	// //position fermeture
	// "DB_BIBLIOTHEQUE".Mobile[#index].Pos[0].Entr0_Ap_Pos[0] := "I_RPO_VER_MLG2";
	// "DB_BIBLIOTHEQUE".Mobile[#index].Pos[0].Entr1_Ap_Pos[0] := "I_RPF_VER_MLG2";
	// "DB_BIBLIOTHEQUE".Mobile[#index].Pos[0].Sort0[0] := "I_CO_ver_MLG2";
	// "DB_BIBLIOTHEQUE".Mobile[#index].Pos[0].Sort0_Pr_Fin_Pos[0] := "I_CO_ver_MLG2";

	// //position ouverture
	// "DB_BIBLIOTHEQUE".Mobile[#index].Pos[1].Entr0_Ap_Pos[0] := "I_RPF_VER_MLG2";
	// "DB_BIBLIOTHEQUE".Mobile[#index].Pos[1].Entr1_Ap_Pos[0] := "I_RPO_VER_MLG2";
	// "DB_BIBLIOTHEQUE".Mobile[#index].Pos[1].Sort1[0] := "I_CO_ver_MLG2";
	// "DB_BIBLIOTHEQUE".Mobile[#index].Pos[1].Sort0_Pr_Fin_Pos[0] := "I_CO_ver_MLG2";
	#index := #index + 1;
	//++++++++++++++++++++++++++++++++++++++++++++++++++++++++++++++/*347*/
	"DB_BIBLIOTHEQUE".Mobile[#index].Nom := 'TMEL2';
	"DB_BIBLIOTHEQUE".Mobile[#index].Tjr_Desasservi := TRUE;
	"Init_Tps"(#index);
	#index := #index + 1;
	//++++++++++++++++++++++++++++++++++++++++++++++++++++++++++++++/*348*/
	"DB_BIBLIOTHEQUE".Mobile[#index].Nom := 'BDBP4';
	"DB_BIBLIOTHEQUE".Mobile[#index].Noeud := TRUE;
	"DB_BIBLIOTHEQUE".Mobile[#index].Mob_Suiv[0] := "Index_Mobile"('MLG1');
	"DB_BIBLIOTHEQUE".Mobile[#index].Mob_Suiv[1] := "Index_Mobile"('MLG2');
	"DB_BIBLIOTHEQUE".Mobile[#index].Pos[0].Nom := 'GAUCHE';
	"DB_BIBLIOTHEQUE".Mobile[#index].Pos[0].Mob_Suiv[0] := "Index_Mobile"('MLG2');
	"DB_BIBLIOTHEQUE".Mobile[#index].Pos[1].Nom := 'DROITE';
	"DB_BIBLIOTHEQUE".Mobile[#index].Pos[1].Mob_Suiv[0] := "Index_Mobile"('MLG');
	"DB_BIBLIOTHEQUE".Mobile[#index].Tjr_Desasservi := TRUE;
	"DB_BIBLIOTHEQUE".Mobile[#index].Tps_Att := t#500ms;
	"DB_BIBLIOTHEQUE".Mobile[#index].Tps_Arr := t#0ms;

	//Entrées
	"DB_BIBLIOTHEQUE".Mobile[#index].Pos[0].Entr0_Ap_Pos[0] := "I_RP_BDBP4_MLG2";
	"DB_BIBLIOTHEQUE".Mobile[#index].Pos[0].Entr1_Ap_Pos[0] := "I_RP_BDBP4_MLG1";
	"DB_BIBLIOTHEQUE".Mobile[#index].Pos[0].Sort1[0] := "I_CP_BDBP4_MLG1";
	"DB_BIBLIOTHEQUE".Mobile[#index].Pos[0].Sort0[0] := "I_CP_BDBP4_MLG2";
	"DB_BIBLIOTHEQUE".Mobile[#index].Pos[0].Sort0_Pr_Fin_Pos[0] := "I_CP_BDBP4_MLG1";
	"DB_BIBLIOTHEQUE".Mobile[#index].Pos[0].Sort0_Pr_Fin_Pos[1] := "I_CP_BDBP4_MLG2";


	"DB_BIBLIOTHEQUE".Mobile[#index].Pos[1].Entr0_Ap_Pos[1] := "I_RP_BDBP4_MLG1";
	"DB_BIBLIOTHEQUE".Mobile[#index].Pos[1].Entr1_Ap_Pos[1] := "I_RP_BDBP4_MLG2";

	//Sorties
	"DB_BIBLIOTHEQUE".Mobile[#index].Pos[1].Sort1[0] := "I_CP_BDBP4_MLG2";
	"DB_BIBLIOTHEQUE".Mobile[#index].Pos[1].Sort0[0] := "I_CP_BDBP4_MLG1";
	"DB_BIBLIOTHEQUE".Mobile[#index].Pos[1].Sort0_Pr_Fin_Pos[0] := "I_CP_BDBP4_MLG1";
	"DB_BIBLIOTHEQUE".Mobile[#index].Pos[1].Sort0_Pr_Fin_Pos[1] := "I_CP_BDBP4_MLG2";
	#index := #index + 1;
	//++++++++++++++++++++++++++++++++++++++++++++++++++++++++++++++/*349*/
	"DB_BIBLIOTHEQUE".Mobile[#index].Nom := 'TRP1_TMEL2';
	// "DB_BIBLIOTHEQUE".Mobile[#index].Mob_Suiv[0] := "Index_Mobile"('TMEL');
	"DB_BIBLIOTHEQUE".Mobile[#index].Pos[0].Nom := 'OUVERTURE';
	"DB_BIBLIOTHEQUE".Mobile[#index].Pos[1].Nom := 'FERMETURE';
	"DB_BIBLIOTHEQUE".Mobile[#index].Tjr_Desasservi := TRUE;
	"Init_Tps"(#index);

	//position fermeture
	"DB_BIBLIOTHEQUE".Mobile[#index].Pos[0].Entr0_Ap_Pos[0] := "I_RPO_TRP1_TMEL2";
	"DB_BIBLIOTHEQUE".Mobile[#index].Pos[0].Entr1_Ap_Pos[0] := "I_RPF_TRP1_TMEL2";
	"DB_BIBLIOTHEQUE".Mobile[#index].Pos[0].Sort0[0] := "I_CO_TRP1_TMEL2";
	"DB_BIBLIOTHEQUE".Mobile[#index].Pos[0].Sort0_Pr_Fin_Pos[0] := "I_CO_TRP1_TMEL2";

	//position ouverture
	"DB_BIBLIOTHEQUE".Mobile[#index].Pos[1].Entr0_Ap_Pos[0] := "I_RPF_TRP1_TMEL2";
	"DB_BIBLIOTHEQUE".Mobile[#index].Pos[1].Entr1_Ap_Pos[0] := "I_RPO_TRP1_TMEL2";
	"DB_BIBLIOTHEQUE".Mobile[#index].Pos[1].Sort1[0] := "I_CO_TRP1_TMEL2";
	"DB_BIBLIOTHEQUE".Mobile[#index].Pos[1].Sort0_Pr_Fin_Pos[0] := "I_CO_TRP1_TMEL2";
	#index := #index + 1;

	//++++++++++++++++++++++++++++++//DD01//++++++++++++++++++++++++++++++++/*350*/
	"DB_BIBLIOTHEQUE".Mobile[#index].Noeud := TRUE;


	"DB_BIBLIOTHEQUE".Mobile[#index].Nom := 'DD01';                                  //NOEUD
	"DB_BIBLIOTHEQUE".Mobile[#index].Mob_Suiv[0] := "Index_Mobile"('BV01');
	"DB_BIBLIOTHEQUE".Mobile[#index].Mob_Suiv[1] := "Index_Mobile"('BV02');
	"DB_BIBLIOTHEQUE".Mobile[#index].Mob_Suiv[2] := "Index_Mobile"('BV03');
	"DB_BIBLIOTHEQUE".Mobile[#index].Mob_Suiv[3] := "Index_Mobile"('BV04');
	"DB_BIBLIOTHEQUE".Mobile[#index].Mob_Suiv[4] := "Index_Mobile"('BV05');
	"DB_BIBLIOTHEQUE".Mobile[#index].Mob_Suiv[5] := "Index_Mobile"('BV06');
	"DB_BIBLIOTHEQUE".Mobile[#index].Mob_Prec[0] := "Index_Mobile"('BDE24');


	"DB_BIBLIOTHEQUE".Mobile[#index].Pos[0].Nom := '_BV01';
	"DB_BIBLIOTHEQUE".Mobile[#index].Pos[0].Mob_Suiv[0] := "Index_Mobile"('BV01');
	"DB_BIBLIOTHEQUE".Mobile[#index].Pos[1].Nom := '_BV02';
	"DB_BIBLIOTHEQUE".Mobile[#index].Pos[1].Mob_Suiv[0] := "Index_Mobile"('BV02');
	"DB_BIBLIOTHEQUE".Mobile[#index].Pos[2].Nom := '_BV03';
	"DB_BIBLIOTHEQUE".Mobile[#index].Pos[2].Mob_Suiv[0] := "Index_Mobile"('BV03');
	"DB_BIBLIOTHEQUE".Mobile[#index].Pos[3].Nom := '_BV04';
	"DB_BIBLIOTHEQUE".Mobile[#index].Pos[3].Mob_Suiv[0] := "Index_Mobile"('BV04');
	"DB_BIBLIOTHEQUE".Mobile[#index].Pos[4].Nom := '_BV05';
	"DB_BIBLIOTHEQUE".Mobile[#index].Pos[4].Mob_Suiv[0] := "Index_Mobile"('BV05');
	"DB_BIBLIOTHEQUE".Mobile[#index].Pos[5].Nom := '_BV06';
	"DB_BIBLIOTHEQUE".Mobile[#index].Pos[5].Mob_Suiv[0] := "Index_Mobile"('BV06');

	"Init_Tps"(#index);

	// VERS BV1
	"DB_BIBLIOTHEQUE".Mobile[#index].Pos[0].Entr0_Ap_Pos[0] := "I_RP_DD01_BV2";
	"DB_BIBLIOTHEQUE".Mobile[#index].Pos[0].Entr0_Ap_Pos[1] := "I_RP_DD01_BV3";
	"DB_BIBLIOTHEQUE".Mobile[#index].Pos[0].Entr0_Ap_Pos[2] := "I_RP_DD01_BV4";
	"DB_BIBLIOTHEQUE".Mobile[#index].Pos[0].Entr0_Ap_Pos[3] := "I_RP_DD01_BV5";
	"DB_BIBLIOTHEQUE".Mobile[#index].Pos[0].Entr0_Ap_Pos[4] := "I_RP_DD01_BV6";
	"DB_BIBLIOTHEQUE".Mobile[#index].Pos[0].Entr1_Ap_Pos[0] := "I_RP_DD01_BV1";
	"DB_BIBLIOTHEQUE".Mobile[#index].Pos[0].Sort1[0] := "I_CM_DD01";
	"DB_BIBLIOTHEQUE".Mobile[#index].Pos[0].Sort1[1] := "I_FCP_DD01_BV1";
	"DB_BIBLIOTHEQUE".Mobile[#index].Pos[0].Sort0_Pr_Fin_Pos[0] := "I_CM_DD01";
	"DB_BIBLIOTHEQUE".Mobile[#index].Pos[0].Sort0_Pr_Fin_Pos[1] := "I_FCP_DD01_BV1";
	"DB_BIBLIOTHEQUE".Mobile[#index].Pos[0].Sort0_Ap_Pos[0] := "I_CM_DD01";
	// VERS BV2
	"DB_BIBLIOTHEQUE".Mobile[#index].Pos[1].Entr0_Ap_Pos[0] := "I_RP_DD01_BV1";
	"DB_BIBLIOTHEQUE".Mobile[#index].Pos[1].Entr0_Ap_Pos[1] := "I_RP_DD01_BV3";
	"DB_BIBLIOTHEQUE".Mobile[#index].Pos[1].Entr0_Ap_Pos[2] := "I_RP_DD01_BV4";
	"DB_BIBLIOTHEQUE".Mobile[#index].Pos[1].Entr0_Ap_Pos[3] := "I_RP_DD01_BV5";
	"DB_BIBLIOTHEQUE".Mobile[#index].Pos[1].Entr0_Ap_Pos[4] := "I_RP_DD01_BV6";
	"DB_BIBLIOTHEQUE".Mobile[#index].Pos[1].Entr1_Ap_Pos[0] := "I_RP_DD01_BV2";
	"DB_BIBLIOTHEQUE".Mobile[#index].Pos[1].Sort1[0] := "I_CM_DD01";
	"DB_BIBLIOTHEQUE".Mobile[#index].Pos[1].Sort1[1] := "I_FCP_DD01_BV2";
	"DB_BIBLIOTHEQUE".Mobile[#index].Pos[1].Sort0_Pr_Fin_Pos[0] := "I_CM_DD01";
	"DB_BIBLIOTHEQUE".Mobile[#index].Pos[1].Sort0_Pr_Fin_Pos[1] := "I_FCP_DD01_BV2";
	"DB_BIBLIOTHEQUE".Mobile[#index].Pos[1].Sort0_Ap_Pos[0] := "I_CM_DD01";
	//VERS BV3
	"DB_BIBLIOTHEQUE".Mobile[#index].Pos[2].Entr0_Ap_Pos[0] := "I_RP_DD01_BV1";
	"DB_BIBLIOTHEQUE".Mobile[#index].Pos[2].Entr0_Ap_Pos[1] := "I_RP_DD01_BV2";
	"DB_BIBLIOTHEQUE".Mobile[#index].Pos[2].Entr0_Ap_Pos[2] := "I_RP_DD01_BV4";
	"DB_BIBLIOTHEQUE".Mobile[#index].Pos[2].Entr0_Ap_Pos[3] := "I_RP_DD01_BV5";
	"DB_BIBLIOTHEQUE".Mobile[#index].Pos[2].Entr0_Ap_Pos[4] := "I_RP_DD01_BV6";
	"DB_BIBLIOTHEQUE".Mobile[#index].Pos[2].Entr1_Ap_Pos[0] := "I_RP_DD01_BV3";
	"DB_BIBLIOTHEQUE".Mobile[#index].Pos[2].Sort1[0] := "I_CM_DD01";
	"DB_BIBLIOTHEQUE".Mobile[#index].Pos[2].Sort1[1] := "I_FCP_DD01_BV3";
	"DB_BIBLIOTHEQUE".Mobile[#index].Pos[2].Sort0_Pr_Fin_Pos[0] := "I_CM_DD01";
	"DB_BIBLIOTHEQUE".Mobile[#index].Pos[2].Sort0_Pr_Fin_Pos[1] := "I_FCP_DD01_BV3";
	"DB_BIBLIOTHEQUE".Mobile[#index].Pos[2].Sort0_Ap_Pos[0] := "I_CM_DD01";
	//VERS BV4
	"DB_BIBLIOTHEQUE".Mobile[#index].Pos[3].Entr0_Ap_Pos[0] := "I_RP_DD01_BV1";
	"DB_BIBLIOTHEQUE".Mobile[#index].Pos[3].Entr0_Ap_Pos[1] := "I_RP_DD01_BV2";
	"DB_BIBLIOTHEQUE".Mobile[#index].Pos[3].Entr0_Ap_Pos[2] := "I_RP_DD01_BV3";
	"DB_BIBLIOTHEQUE".Mobile[#index].Pos[3].Entr0_Ap_Pos[3] := "I_RP_DD01_BV5";
	"DB_BIBLIOTHEQUE".Mobile[#index].Pos[3].Entr0_Ap_Pos[4] := "I_RP_DD01_BV6";
	"DB_BIBLIOTHEQUE".Mobile[#index].Pos[3].Entr1_Ap_Pos[0] := "I_RP_DD01_BV4";
	"DB_BIBLIOTHEQUE".Mobile[#index].Pos[3].Sort1[0] := "I_CM_DD01";
	"DB_BIBLIOTHEQUE".Mobile[#index].Pos[3].Sort1[1] := "I_FCP_DD01_BV4";
	"DB_BIBLIOTHEQUE".Mobile[#index].Pos[3].Sort0_Pr_Fin_Pos[0] := "I_CM_DD01";
	"DB_BIBLIOTHEQUE".Mobile[#index].Pos[3].Sort0_Pr_Fin_Pos[1] := "I_FCP_DD01_BV4";
	"DB_BIBLIOTHEQUE".Mobile[#index].Pos[3].Sort0_Ap_Pos[0] := "I_CM_DD01";
	//VERS BV5
	"DB_BIBLIOTHEQUE".Mobile[#index].Pos[4].Entr0_Ap_Pos[0] := "I_RP_DD01_BV1";
	"DB_BIBLIOTHEQUE".Mobile[#index].Pos[4].Entr0_Ap_Pos[1] := "I_RP_DD01_BV2";
	"DB_BIBLIOTHEQUE".Mobile[#index].Pos[4].Entr0_Ap_Pos[2] := "I_RP_DD01_BV3";
	"DB_BIBLIOTHEQUE".Mobile[#index].Pos[4].Entr0_Ap_Pos[3] := "I_RP_DD01_BV4";
	"DB_BIBLIOTHEQUE".Mobile[#index].Pos[4].Entr0_Ap_Pos[4] := "I_RP_DD01_BV6";
	"DB_BIBLIOTHEQUE".Mobile[#index].Pos[4].Entr1_Ap_Pos[0] := "I_RP_DD01_BV5";
	"DB_BIBLIOTHEQUE".Mobile[#index].Pos[4].Sort1[0] := "I_CM_DD01";
	"DB_BIBLIOTHEQUE".Mobile[#index].Pos[4].Sort1[1] := "I_FCP_DD01_BV5";
	"DB_BIBLIOTHEQUE".Mobile[#index].Pos[4].Sort0_Pr_Fin_Pos[0] := "I_CM_DD01";
	"DB_BIBLIOTHEQUE".Mobile[#index].Pos[4].Sort0_Pr_Fin_Pos[1] := "I_FCP_DD01_BV5";
	"DB_BIBLIOTHEQUE".Mobile[#index].Pos[4].Sort0_Ap_Pos[0] := "I_CM_DD01";
	//VERS BV6
	"DB_BIBLIOTHEQUE".Mobile[#index].Pos[5].Entr0_Ap_Pos[0] := "I_RP_DD01_BV1";
	"DB_BIBLIOTHEQUE".Mobile[#index].Pos[5].Entr0_Ap_Pos[1] := "I_RP_DD01_BV2";
	"DB_BIBLIOTHEQUE".Mobile[#index].Pos[5].Entr0_Ap_Pos[2] := "I_RP_DD01_BV3";
	"DB_BIBLIOTHEQUE".Mobile[#index].Pos[5].Entr0_Ap_Pos[3] := "I_RP_DD01_BV4";
	"DB_BIBLIOTHEQUE".Mobile[#index].Pos[5].Entr0_Ap_Pos[4] := "I_RP_DD01_BV5";
	"DB_BIBLIOTHEQUE".Mobile[#index].Pos[5].Entr1_Ap_Pos[0] := "I_RP_DD01_BV6";
	"DB_BIBLIOTHEQUE".Mobile[#index].Pos[5].Sort1[0] := "I_CM_DD01";
	"DB_BIBLIOTHEQUE".Mobile[#index].Pos[5].Sort1[1] := "I_FCP_DD01_BV6";
	"DB_BIBLIOTHEQUE".Mobile[#index].Pos[5].Sort0_Pr_Fin_Pos[0] := "I_CM_DD01";
	"DB_BIBLIOTHEQUE".Mobile[#index].Pos[5].Sort0_Pr_Fin_Pos[1] := "I_FCP_DD01_BV6";
	"DB_BIBLIOTHEQUE".Mobile[#index].Pos[5].Sort0_Ap_Pos[0] := "I_CM_DD01";
	#index := #index + 1;
	//++++++++++++++++++++++++++++++//DD02//++++++++++++++++++++++++++++++++/*351*/
	"DB_BIBLIOTHEQUE".Mobile[#index].Nom := 'DD02';
	"DB_BIBLIOTHEQUE".Mobile[#index].Noeud := TRUE;  //NOEUD
	"DB_BIBLIOTHEQUE".Mobile[#index].Mob_Suiv[0] := "Index_Mobile"('BV07');
	"DB_BIBLIOTHEQUE".Mobile[#index].Mob_Suiv[1] := "Index_Mobile"('BV08');
	"DB_BIBLIOTHEQUE".Mobile[#index].Mob_Suiv[2] := "Index_Mobile"('BV09');
	"DB_BIBLIOTHEQUE".Mobile[#index].Mob_Suiv[3] := "Index_Mobile"('BV10');
	"DB_BIBLIOTHEQUE".Mobile[#index].Mob_Suiv[4] := "Index_Mobile"('BV11');
	"DB_BIBLIOTHEQUE".Mobile[#index].Mob_Suiv[5] := "Index_Mobile"('BV12');
	"DB_BIBLIOTHEQUE".Mobile[#index].Mob_Prec[0] := "Index_Mobile"('T54');

	"DB_BIBLIOTHEQUE".Mobile[#index].Pos[0].Nom := '_BV07';
	"DB_BIBLIOTHEQUE".Mobile[#index].Pos[0].Mob_Suiv[0] := "Index_Mobile"('BV07');
	"DB_BIBLIOTHEQUE".Mobile[#index].Pos[1].Nom := '_BV08';
	"DB_BIBLIOTHEQUE".Mobile[#index].Pos[1].Mob_Suiv[0] := "Index_Mobile"('BV08');
	"DB_BIBLIOTHEQUE".Mobile[#index].Pos[2].Nom := '_BV09';
	"DB_BIBLIOTHEQUE".Mobile[#index].Pos[2].Mob_Suiv[0] := "Index_Mobile"('BV09');
	"DB_BIBLIOTHEQUE".Mobile[#index].Pos[3].Nom := '_BV10';
	"DB_BIBLIOTHEQUE".Mobile[#index].Pos[3].Mob_Suiv[0] := "Index_Mobile"('BV10');
	"DB_BIBLIOTHEQUE".Mobile[#index].Pos[4].Nom := '_BV11';
	"DB_BIBLIOTHEQUE".Mobile[#index].Pos[4].Mob_Suiv[0] := "Index_Mobile"('BV11');
	"DB_BIBLIOTHEQUE".Mobile[#index].Pos[5].Nom := '_BV12';
	"DB_BIBLIOTHEQUE".Mobile[#index].Pos[5].Mob_Suiv[0] := "Index_Mobile"('BV12');

	"Init_Tps"(#index);


	// VERS BV7
	"DB_BIBLIOTHEQUE".Mobile[#index].Pos[0].Entr0_Ap_Pos[0] := "I_RP_DD02_BV8";
	"DB_BIBLIOTHEQUE".Mobile[#index].Pos[0].Entr0_Ap_Pos[1] := "I_RP_DD02_BV9";
	"DB_BIBLIOTHEQUE".Mobile[#index].Pos[0].Entr0_Ap_Pos[2] := "I_RP_DD02_BV10";
	"DB_BIBLIOTHEQUE".Mobile[#index].Pos[0].Entr0_Ap_Pos[3] := "I_RP_DD02_BV11";
	"DB_BIBLIOTHEQUE".Mobile[#index].Pos[0].Entr0_Ap_Pos[4] := "I_RP_DD02_BV12";
	"DB_BIBLIOTHEQUE".Mobile[#index].Pos[0].Entr1_Ap_Pos[0] := "I_RP_DD02_BV7";
	"DB_BIBLIOTHEQUE".Mobile[#index].Pos[0].Sort1[0] := "I_CM_DD02";
	"DB_BIBLIOTHEQUE".Mobile[#index].Pos[0].Sort1[1] := "I_FCP_DD02_BV7";
	"DB_BIBLIOTHEQUE".Mobile[#index].Pos[0].Sort0_Pr_Fin_Pos[0] := "I_CM_DD02";
	"DB_BIBLIOTHEQUE".Mobile[#index].Pos[0].Sort0_Pr_Fin_Pos[1] := "I_FCP_DD02_BV7";
	"DB_BIBLIOTHEQUE".Mobile[#index].Pos[0].Sort0_Ap_Pos[0] := "I_CM_DD02";
	// VERS BV8
	"DB_BIBLIOTHEQUE".Mobile[#index].Pos[1].Entr0_Ap_Pos[0] := "I_RP_DD02_BV7";
	"DB_BIBLIOTHEQUE".Mobile[#index].Pos[1].Entr0_Ap_Pos[1] := "I_RP_DD02_BV9";
	"DB_BIBLIOTHEQUE".Mobile[#index].Pos[1].Entr0_Ap_Pos[2] := "I_RP_DD02_BV10";
	"DB_BIBLIOTHEQUE".Mobile[#index].Pos[1].Entr0_Ap_Pos[3] := "I_RP_DD02_BV11";
	"DB_BIBLIOTHEQUE".Mobile[#index].Pos[1].Entr0_Ap_Pos[4] := "I_RP_DD02_BV12";
	"DB_BIBLIOTHEQUE".Mobile[#index].Pos[1].Entr1_Ap_Pos[0] := "I_RP_DD02_BV8";
	"DB_BIBLIOTHEQUE".Mobile[#index].Pos[1].Sort1[0] := "I_CM_DD02";
	"DB_BIBLIOTHEQUE".Mobile[#index].Pos[1].Sort1[1] := "I_FCP_DD02_BV8";
	"DB_BIBLIOTHEQUE".Mobile[#index].Pos[1].Sort0_Pr_Fin_Pos[0] := "I_CM_DD02";
	"DB_BIBLIOTHEQUE".Mobile[#index].Pos[1].Sort0_Pr_Fin_Pos[1] := "I_FCP_DD02_BV8";
	"DB_BIBLIOTHEQUE".Mobile[#index].Pos[1].Sort0_Ap_Pos[0] := "I_CM_DD02";
	//VERS BV9
	"DB_BIBLIOTHEQUE".Mobile[#index].Pos[2].Entr0_Ap_Pos[0] := "I_RP_DD02_BV7";
	"DB_BIBLIOTHEQUE".Mobile[#index].Pos[2].Entr0_Ap_Pos[1] := "I_RP_DD02_BV8";
	"DB_BIBLIOTHEQUE".Mobile[#index].Pos[2].Entr0_Ap_Pos[2] := "I_RP_DD02_BV10";
	"DB_BIBLIOTHEQUE".Mobile[#index].Pos[2].Entr0_Ap_Pos[3] := "I_RP_DD02_BV11";
	"DB_BIBLIOTHEQUE".Mobile[#index].Pos[2].Entr0_Ap_Pos[4] := "I_RP_DD02_BV12";
	"DB_BIBLIOTHEQUE".Mobile[#index].Pos[2].Entr1_Ap_Pos[0] := "I_RP_DD02_BV9";
	"DB_BIBLIOTHEQUE".Mobile[#index].Pos[2].Sort1[0] := "I_CM_DD02";
	"DB_BIBLIOTHEQUE".Mobile[#index].Pos[2].Sort1[1] := "I_FCP_DD02_BV9";
	"DB_BIBLIOTHEQUE".Mobile[#index].Pos[2].Sort0_Pr_Fin_Pos[0] := "I_CM_DD02";
	"DB_BIBLIOTHEQUE".Mobile[#index].Pos[2].Sort0_Pr_Fin_Pos[1] := "I_FCP_DD02_BV9";
	"DB_BIBLIOTHEQUE".Mobile[#index].Pos[2].Sort0_Ap_Pos[0] := "I_CM_DD02";
	//VERS BV10
	"DB_BIBLIOTHEQUE".Mobile[#index].Pos[3].Entr0_Ap_Pos[0] := "I_RP_DD02_BV7";
	"DB_BIBLIOTHEQUE".Mobile[#index].Pos[3].Entr0_Ap_Pos[1] := "I_RP_DD02_BV8";
	"DB_BIBLIOTHEQUE".Mobile[#index].Pos[3].Entr0_Ap_Pos[2] := "I_RP_DD02_BV9";
	"DB_BIBLIOTHEQUE".Mobile[#index].Pos[3].Entr0_Ap_Pos[3] := "I_RP_DD02_BV11";
	"DB_BIBLIOTHEQUE".Mobile[#index].Pos[3].Entr0_Ap_Pos[4] := "I_RP_DD02_BV12";
	"DB_BIBLIOTHEQUE".Mobile[#index].Pos[3].Entr1_Ap_Pos[0] := "I_RP_DD02_BV10";
	"DB_BIBLIOTHEQUE".Mobile[#index].Pos[3].Sort1[0] := "I_CM_DD02";
	"DB_BIBLIOTHEQUE".Mobile[#index].Pos[3].Sort1[1] := "I_FCP_DD02_BV10";
	"DB_BIBLIOTHEQUE".Mobile[#index].Pos[3].Sort0_Pr_Fin_Pos[0] := "I_CM_DD02";
	"DB_BIBLIOTHEQUE".Mobile[#index].Pos[3].Sort0_Pr_Fin_Pos[1] := "I_FCP_DD02_BV10";
	"DB_BIBLIOTHEQUE".Mobile[#index].Pos[3].Sort0_Ap_Pos[0] := "I_CM_DD02";
	//VERS BV11
	"DB_BIBLIOTHEQUE".Mobile[#index].Pos[4].Entr0_Ap_Pos[0] := "I_RP_DD02_BV7";
	"DB_BIBLIOTHEQUE".Mobile[#index].Pos[4].Entr0_Ap_Pos[1] := "I_RP_DD02_BV8";
	"DB_BIBLIOTHEQUE".Mobile[#index].Pos[4].Entr0_Ap_Pos[2] := "I_RP_DD02_BV9";
	"DB_BIBLIOTHEQUE".Mobile[#index].Pos[4].Entr0_Ap_Pos[3] := "I_RP_DD02_BV10";
	"DB_BIBLIOTHEQUE".Mobile[#index].Pos[4].Entr0_Ap_Pos[4] := "I_RP_DD02_BV12";
	"DB_BIBLIOTHEQUE".Mobile[#index].Pos[4].Entr1_Ap_Pos[0] := "I_RP_DD02_BV11";
	"DB_BIBLIOTHEQUE".Mobile[#index].Pos[4].Sort1[0] := "I_CM_DD02";
	"DB_BIBLIOTHEQUE".Mobile[#index].Pos[4].Sort1[1] := "I_FCP_DD02_BV11";
	"DB_BIBLIOTHEQUE".Mobile[#index].Pos[4].Sort0_Pr_Fin_Pos[0] := "I_CM_DD02";
	"DB_BIBLIOTHEQUE".Mobile[#index].Pos[4].Sort0_Pr_Fin_Pos[1] := "I_FCP_DD02_BV11";
	"DB_BIBLIOTHEQUE".Mobile[#index].Pos[4].Sort0_Ap_Pos[0] := "I_CM_DD02";
	//VERS BV12
	"DB_BIBLIOTHEQUE".Mobile[#index].Pos[5].Entr0_Ap_Pos[0] := "I_RP_DD02_BV7";
	"DB_BIBLIOTHEQUE".Mobile[#index].Pos[5].Entr0_Ap_Pos[1] := "I_RP_DD02_BV8";
	"DB_BIBLIOTHEQUE".Mobile[#index].Pos[5].Entr0_Ap_Pos[2] := "I_RP_DD02_BV9";
	"DB_BIBLIOTHEQUE".Mobile[#index].Pos[5].Entr0_Ap_Pos[3] := "I_RP_DD02_BV10";
	"DB_BIBLIOTHEQUE".Mobile[#index].Pos[5].Entr0_Ap_Pos[4] := "I_RP_DD02_BV11";
	"DB_BIBLIOTHEQUE".Mobile[#index].Pos[5].Entr1_Ap_Pos[0] := "I_RP_DD02_BV12";
	"DB_BIBLIOTHEQUE".Mobile[#index].Pos[5].Sort1[0] := "I_CM_DD02";
	"DB_BIBLIOTHEQUE".Mobile[#index].Pos[5].Sort1[1] := "I_FCP_DD02_BV12";
	"DB_BIBLIOTHEQUE".Mobile[#index].Pos[5].Sort0_Pr_Fin_Pos[0] := "I_CM_DD02";
	"DB_BIBLIOTHEQUE".Mobile[#index].Pos[5].Sort0_Pr_Fin_Pos[1] := "I_FCP_DD02_BV12";
	"DB_BIBLIOTHEQUE".Mobile[#index].Pos[5].Sort0_Ap_Pos[0] := "I_CM_DD02";
	#index := #index + 1;
	//++++++++++++++++++++++++++++++//ORIGINE FICTIF POUR EXPEDITION//++++++++++++++++++++++++++++++++/*352*/
	"DB_BIBLIOTHEQUE".Mobile[#index].Nom := 'O_Exp_Fict';
	"DB_BIBLIOTHEQUE".Mobile[#index].Mob_Suiv[0] := "Index_Mobile"('E12');
	"DB_BIBLIOTHEQUE".Mobile[#index].Pos[0].Nom := 'VERS_E12';
	"DB_BIBLIOTHEQUE".Mobile[#index].Pos[0].Mob_Suiv[0] := "Index_Mobile"('E12');
	"DB_BIBLIOTHEQUE".Mobile[#index].Tps_Att := t#500ms;
	"DB_BIBLIOTHEQUE".Mobile[#index].Tps_Arr := t#0ms;
	#index := #index + 1;
	//++++++++++++++++++++++++++++++++++++++++++++++++++++++++++++++/*353*/
	"DB_BIBLIOTHEQUE".Mobile[#index].Nom := 'BP03';
	"DB_BIBLIOTHEQUE".Mobile[#index].Pos[0].Nom := 'Vid';
	"DB_BIBLIOTHEQUE".Mobile[#index].Tjr_Desasservi := TRUE;
	"Init_Tps"(#index);
	#index := #index + 1;
	//++++++++++++++++++++++++++++++++++++++++++++++++++++++++++++++/*354*/
	"DB_BIBLIOTHEQUE".Mobile[#index].Nom := 'BDVS';
	"DB_BIBLIOTHEQUE".Mobile[#index].Noeud := TRUE;
	"DB_BIBLIOTHEQUE".Mobile[#index].Mob_Suiv[0] := "Index_Mobile"('MLG2');
	"DB_BIBLIOTHEQUE".Mobile[#index].Mob_Suiv[1] := "Index_Mobile"('MLG1');
	"DB_BIBLIOTHEQUE".Mobile[#index].Pos[0].Nom := 'VERS_MLG2';
	"DB_BIBLIOTHEQUE".Mobile[#index].Pos[1].Nom := 'VERS_MLG1';
	"DB_BIBLIOTHEQUE".Mobile[#index].Tjr_Desasservi := TRUE;

	//Entrées
	"DB_BIBLIOTHEQUE".Mobile[#index].Pos[0].Entr0_Ap_Pos[0] := "I_RP_BDVS_MLG1";
	"DB_BIBLIOTHEQUE".Mobile[#index].Pos[0].Entr1_Ap_Pos[0] := "I_RP_BDVS_MLG2";
	//Sorties
	"DB_BIBLIOTHEQUE".Mobile[#index].Pos[0].Sort1[0] := "I_CP_BDVS_MLG2";
	"DB_BIBLIOTHEQUE".Mobile[#index].Pos[0].Sort0[0] := "I_CP_BDVS_MLG1";
	"DB_BIBLIOTHEQUE".Mobile[#index].Pos[0].Sort0_Pr_Fin_Pos[0] := "I_CP_BDVS_MLG1";
	"DB_BIBLIOTHEQUE".Mobile[#index].Pos[0].Sort0_Pr_Fin_Pos[1] := "I_CP_BDVS_MLG2";

	//Entrées
	"DB_BIBLIOTHEQUE".Mobile[#index].Pos[1].Entr0_Ap_Pos[1] := "I_RP_BDVS_MLG2";
	"DB_BIBLIOTHEQUE".Mobile[#index].Pos[1].Entr1_Ap_Pos[1] := "I_RP_BDVS_MLG1";
	//Sorties
	"DB_BIBLIOTHEQUE".Mobile[#index].Pos[1].Sort1[0] := "I_CP_BDVS_MLG1";
	"DB_BIBLIOTHEQUE".Mobile[#index].Pos[1].Sort0[0] := "I_CP_BDVS_MLG2";
	"DB_BIBLIOTHEQUE".Mobile[#index].Pos[1].Sort0_Pr_Fin_Pos[0] := "I_CP_BDVS_MLG1";
	"DB_BIBLIOTHEQUE".Mobile[#index].Pos[1].Sort0_Pr_Fin_Pos[1] := "I_CP_BDVS_MLG2";
	"Init_Tps"(#index);
	#index := #index + 1;
	//++++++++++++++++++++++++++++++++++++++++++++++++++++++++++++++/*355*/
	"DB_BIBLIOTHEQUE".Mobile[#index].Nom := 'TRP_VID_VS';
	"DB_BIBLIOTHEQUE".Mobile[#index].Pos[0].Nom := 'FERMETURE';
	"DB_BIBLIOTHEQUE".Mobile[#index].Pos[1].Nom := 'OUVERTURE';
	"DB_BIBLIOTHEQUE".Mobile[#index].Tjr_Desasservi := TRUE;

	//position fermeture
	"DB_BIBLIOTHEQUE".Mobile[#index].Pos[0].Entr0_Ap_Pos[0] := "I_RPO_TRP_VID_VS";
	"DB_BIBLIOTHEQUE".Mobile[#index].Pos[0].Entr1_Ap_Pos[0] := "I_RPF_TRP_VID_VS";
	"DB_BIBLIOTHEQUE".Mobile[#index].Pos[0].Sort0[0] := "I_CO_TRP_VID_VS";
	"DB_BIBLIOTHEQUE".Mobile[#index].Pos[0].Sort0_Pr_Fin_Pos[0] := "I_CO_TRP_VID_VS";

	//position ouverture
	"DB_BIBLIOTHEQUE".Mobile[#index].Pos[1].Entr0_Ap_Pos[0] := "I_RPF_TRP_VID_VS";
	"DB_BIBLIOTHEQUE".Mobile[#index].Pos[1].Entr1_Ap_Pos[0] := "I_RPO_TRP_VID_VS";
	"DB_BIBLIOTHEQUE".Mobile[#index].Pos[1].Sort1[0] := "I_CO_TRP_VID_VS";
	"DB_BIBLIOTHEQUE".Mobile[#index].Pos[1].Sort0_Pr_Fin_Pos[0] := "I_CO_TRP_VID_VS";

	"Init_Tps"(#index);
	#index := #index + 1;
	//++++++++++++++++++++++++++++++++++++++++++++++++++++++++++++++/*356*/
	"DB_BIBLIOTHEQUE".Mobile[#index].Nom := 'TRP_ET_VS';
	"DB_BIBLIOTHEQUE".Mobile[#index].Pos[0].Nom := 'FERMETURE';
	"DB_BIBLIOTHEQUE".Mobile[#index].Pos[1].Nom := 'OUVERTURE';
	"DB_BIBLIOTHEQUE".Mobile[#index].Tjr_Desasservi := TRUE;

	//position fermeture
	"DB_BIBLIOTHEQUE".Mobile[#index].Pos[0].Entr0_Ap_Pos[0] := "I_RPO_TRP_ET_VS";
	"DB_BIBLIOTHEQUE".Mobile[#index].Pos[0].Entr1_Ap_Pos[0] := "I_RPF_TRP_ET_VS";
	"DB_BIBLIOTHEQUE".Mobile[#index].Pos[0].Sort0[0] := "I_CO_TRP_ET_VS";
	"DB_BIBLIOTHEQUE".Mobile[#index].Pos[0].Sort0_Pr_Fin_Pos[0] := "I_CO_TRP_ET_VS";

	//position ouverture
	"DB_BIBLIOTHEQUE".Mobile[#index].Pos[1].Entr0_Ap_Pos[0] := "I_RPF_TRP_ET_VS";
	"DB_BIBLIOTHEQUE".Mobile[#index].Pos[1].Entr1_Ap_Pos[0] := "I_RPO_TRP_ET_VS";
	"DB_BIBLIOTHEQUE".Mobile[#index].Pos[1].Sort1[0] := "I_CO_TRP_ET_VS";
	"DB_BIBLIOTHEQUE".Mobile[#index].Pos[1].Sort0_Pr_Fin_Pos[0] := "I_CO_TRP_ET_VS";

	"Init_Tps"(#index);
	#index := #index + 1;
	//++++++++++++++++++++++++++++++++++++++++++++++++++++++++++++++/*357*/
	"DB_BIBLIOTHEQUE".Mobile[#index].Nom := 'EXT2_S50';
	"DB_BIBLIOTHEQUE".Mobile[#index].Tjr_Desasservi := TRUE;
	"DB_BIBLIOTHEQUE".Mobile[#index].Pos[0].Nom := 'DROIT';
	"Init_Tps"(#index);

	//position fermeture
	"DB_BIBLIOTHEQUE".Mobile[#index].Pos[0].Entr0_Ap_Pos[0] := "I_RPO_TRS50";
	"DB_BIBLIOTHEQUE".Mobile[#index].Pos[0].Entr1_Ap_Pos[0] := "I_RPF_TRS50";
	"DB_BIBLIOTHEQUE".Mobile[#index].Pos[0].Sort0[0] := "I_CO_TRS50";
	"DB_BIBLIOTHEQUE".Mobile[#index].Pos[0].Sort0_Pr_Fin_Pos[0] := "I_CO_TRS50";

	//position ouverture
	"DB_BIBLIOTHEQUE".Mobile[#index].Pos[1].Entr0_Ap_Pos[0] := "I_RPF_TRS50";
	"DB_BIBLIOTHEQUE".Mobile[#index].Pos[1].Entr1_Ap_Pos[0] := "I_RPO_TRS50";
	"DB_BIBLIOTHEQUE".Mobile[#index].Pos[1].Sort1[0] := "I_CO_TRS50";
	"DB_BIBLIOTHEQUE".Mobile[#index].Pos[1].Sort0_Pr_Fin_Pos[0] := "I_CO_TRS50";
	#index := #index + 1;
	//++++++++++++++++++++++++++++++++++++++++++++++++++++++++++++++/*358*/
	"DB_BIBLIOTHEQUE".Mobile[#index].Nom := 'EXT2_S51';
	"DB_BIBLIOTHEQUE".Mobile[#index].Tjr_Desasservi := TRUE;
	"DB_BIBLIOTHEQUE".Mobile[#index].Pos[0].Nom := 'DROIT';
	"Init_Tps"(#index);

	//position fermeture
	"DB_BIBLIOTHEQUE".Mobile[#index].Pos[0].Entr0_Ap_Pos[0] := "I_RPO_TRS51";
	"DB_BIBLIOTHEQUE".Mobile[#index].Pos[0].Entr1_Ap_Pos[0] := "I_RPF_TRS51";
	"DB_BIBLIOTHEQUE".Mobile[#index].Pos[0].Sort0[0] := "I_CO_TRS51";
	"DB_BIBLIOTHEQUE".Mobile[#index].Pos[0].Sort0_Pr_Fin_Pos[0] := "I_CO_TRS51";

	//position ouverture
	"DB_BIBLIOTHEQUE".Mobile[#index].Pos[1].Entr0_Ap_Pos[0] := "I_RPF_TRS51";
	"DB_BIBLIOTHEQUE".Mobile[#index].Pos[1].Entr1_Ap_Pos[0] := "I_RPO_TRS51";
	"DB_BIBLIOTHEQUE".Mobile[#index].Pos[1].Sort1[0] := "I_CO_TRS51";
	"DB_BIBLIOTHEQUE".Mobile[#index].Pos[1].Sort0_Pr_Fin_Pos[0] := "I_CO_TRS51";
	#index := #index + 1;
	//++++++++++++++++++++++++++++++++++++++++++++++++++++++++++++++/*359*/
	"DB_BIBLIOTHEQUE".Mobile[#index].Nom := 'EXT2_S52';
	"DB_BIBLIOTHEQUE".Mobile[#index].Tjr_Desasservi := TRUE;
	"DB_BIBLIOTHEQUE".Mobile[#index].Pos[0].Nom := 'DROIT';
	"Init_Tps"(#index);

	//position fermeture
	"DB_BIBLIOTHEQUE".Mobile[#index].Pos[0].Entr0_Ap_Pos[0] := "I_RPO_TRS52";
	"DB_BIBLIOTHEQUE".Mobile[#index].Pos[0].Entr1_Ap_Pos[0] := "I_RPF_TRS52";
	"DB_BIBLIOTHEQUE".Mobile[#index].Pos[0].Sort0[0] := "I_CO_TRS52";
	"DB_BIBLIOTHEQUE".Mobile[#index].Pos[0].Sort0_Pr_Fin_Pos[0] := "I_CO_TRS52";

	//position ouverture
	"DB_BIBLIOTHEQUE".Mobile[#index].Pos[1].Entr0_Ap_Pos[0] := "I_RPF_TRS52";
	"DB_BIBLIOTHEQUE".Mobile[#index].Pos[1].Entr1_Ap_Pos[0] := "I_RPO_TRS52";
	"DB_BIBLIOTHEQUE".Mobile[#index].Pos[1].Sort1[0] := "I_CO_TRS52";
	"DB_BIBLIOTHEQUE".Mobile[#index].Pos[1].Sort0_Pr_Fin_Pos[0] := "I_CO_TRS52";
	#index := #index + 1;
	//++++++++++++++++++++++++++++++++++++++++++++++++++++++++++++++/*360*/
	"DB_BIBLIOTHEQUE".Mobile[#index].Nom := 'EXT2_S53';
	"DB_BIBLIOTHEQUE".Mobile[#index].Tjr_Desasservi := TRUE;
	"DB_BIBLIOTHEQUE".Mobile[#index].Pos[0].Nom := 'DROIT';
	"Init_Tps"(#index);

	//position fermeture
	"DB_BIBLIOTHEQUE".Mobile[#index].Pos[0].Entr0_Ap_Pos[0] := "I_RPO_TRS53";
	"DB_BIBLIOTHEQUE".Mobile[#index].Pos[0].Entr1_Ap_Pos[0] := "I_RPF_TRS53";
	"DB_BIBLIOTHEQUE".Mobile[#index].Pos[0].Sort0[0] := "I_CO_TRS53";
	"DB_BIBLIOTHEQUE".Mobile[#index].Pos[0].Sort0_Pr_Fin_Pos[0] := "I_CO_TRS53";

	//position ouverture
	"DB_BIBLIOTHEQUE".Mobile[#index].Pos[1].Entr0_Ap_Pos[0] := "I_RPF_TRS53";
	"DB_BIBLIOTHEQUE".Mobile[#index].Pos[1].Entr1_Ap_Pos[0] := "I_RPO_TRS53";
	"DB_BIBLIOTHEQUE".Mobile[#index].Pos[1].Sort1[0] := "I_CO_TRS53";
	"DB_BIBLIOTHEQUE".Mobile[#index].Pos[1].Sort0_Pr_Fin_Pos[0] := "I_CO_TRS53";
	#index := #index + 1;
	//++++++++++++++++++++++++++++++++++++++++++++++++++++++++++++++/*361*/
	"DB_BIBLIOTHEQUE".Mobile[#index].Nom := 'EXT2_S54';
	"DB_BIBLIOTHEQUE".Mobile[#index].Tjr_Desasservi := TRUE;
	"DB_BIBLIOTHEQUE".Mobile[#index].Pos[0].Nom := 'DROIT';
	"Init_Tps"(#index);

	//position fermeture
	"DB_BIBLIOTHEQUE".Mobile[#index].Pos[0].Entr0_Ap_Pos[0] := "I_RPO_TRS54";
	"DB_BIBLIOTHEQUE".Mobile[#index].Pos[0].Entr1_Ap_Pos[0] := "I_RPF_TRS54";
	"DB_BIBLIOTHEQUE".Mobile[#index].Pos[0].Sort0[0] := "I_CO_TRS54";
	"DB_BIBLIOTHEQUE".Mobile[#index].Pos[0].Sort0_Pr_Fin_Pos[0] := "I_CO_TRS54";

	//position ouverture
	"DB_BIBLIOTHEQUE".Mobile[#index].Pos[1].Entr0_Ap_Pos[0] := "I_RPF_TRS54";
	"DB_BIBLIOTHEQUE".Mobile[#index].Pos[1].Entr1_Ap_Pos[0] := "I_RPO_TRS54";
	"DB_BIBLIOTHEQUE".Mobile[#index].Pos[1].Sort1[0] := "I_CO_TRS54";
	"DB_BIBLIOTHEQUE".Mobile[#index].Pos[1].Sort0_Pr_Fin_Pos[0] := "I_CO_TRS54";
	#index := #index + 1;
	//++++++++++++++++++++++++++++++++++++++++++++++++++++++++++++++/*362*/
	"DB_BIBLIOTHEQUE".Mobile[#index].Nom := 'EXT2_S55';
	"DB_BIBLIOTHEQUE".Mobile[#index].Tjr_Desasservi := TRUE;
	"DB_BIBLIOTHEQUE".Mobile[#index].Pos[0].Nom := 'DROIT';
	"Init_Tps"(#index);

	//position fermeture
	"DB_BIBLIOTHEQUE".Mobile[#index].Pos[0].Entr0_Ap_Pos[0] := "I_RPO_TRS55";
	"DB_BIBLIOTHEQUE".Mobile[#index].Pos[0].Entr1_Ap_Pos[0] := "I_RPF_TRS55";
	"DB_BIBLIOTHEQUE".Mobile[#index].Pos[0].Sort0[0] := "I_CO_TRS55";
	"DB_BIBLIOTHEQUE".Mobile[#index].Pos[0].Sort0_Pr_Fin_Pos[0] := "I_CO_TRS55";

	//position ouverture
	"DB_BIBLIOTHEQUE".Mobile[#index].Pos[1].Entr0_Ap_Pos[0] := "I_RPF_TRS55";
	"DB_BIBLIOTHEQUE".Mobile[#index].Pos[1].Entr1_Ap_Pos[0] := "I_RPO_TRS55";
	"DB_BIBLIOTHEQUE".Mobile[#index].Pos[1].Sort1[0] := "I_CO_TRS55";
	"DB_BIBLIOTHEQUE".Mobile[#index].Pos[1].Sort0_Pr_Fin_Pos[0] := "I_CO_TRS55";
	#index := #index + 1;
	//++++++++++++++++++++++++++++++++++++++++++++++++++++++++++++++/*363*/
	"DB_BIBLIOTHEQUE".Mobile[#index].Nom := 'EXT2_S56';
	"DB_BIBLIOTHEQUE".Mobile[#index].Tjr_Desasservi := TRUE;
	"DB_BIBLIOTHEQUE".Mobile[#index].Pos[0].Nom := 'DROIT';
	"Init_Tps"(#index);

	//position fermeture
	"DB_BIBLIOTHEQUE".Mobile[#index].Pos[0].Entr0_Ap_Pos[0] := "I_RPO_TRS56";
	"DB_BIBLIOTHEQUE".Mobile[#index].Pos[0].Entr1_Ap_Pos[0] := "I_RPF_TRS56";
	"DB_BIBLIOTHEQUE".Mobile[#index].Pos[0].Sort0[0] := "I_CO_TRS56";
	"DB_BIBLIOTHEQUE".Mobile[#index].Pos[0].Sort0_Pr_Fin_Pos[0] := "I_CO_TRS56";

	//position ouverture
	"DB_BIBLIOTHEQUE".Mobile[#index].Pos[1].Entr0_Ap_Pos[0] := "I_RPF_TRS56";
	"DB_BIBLIOTHEQUE".Mobile[#index].Pos[1].Entr1_Ap_Pos[0] := "I_RPO_TRS56";
	"DB_BIBLIOTHEQUE".Mobile[#index].Pos[1].Sort1[0] := "I_CO_TRS56";
	"DB_BIBLIOTHEQUE".Mobile[#index].Pos[1].Sort0_Pr_Fin_Pos[0] := "I_CO_TRS56";
	#index := #index + 1;
	//++++++++++++++++++++++++++++++++++++++++++++++++++++++++++++++/*364*/
	"DB_BIBLIOTHEQUE".Mobile[#index].Nom := 'EXT2_S57';
	"DB_BIBLIOTHEQUE".Mobile[#index].Tjr_Desasservi := TRUE;
	"DB_BIBLIOTHEQUE".Mobile[#index].Pos[0].Nom := 'DROIT';
	"Init_Tps"(#index);

	//position fermeture
	"DB_BIBLIOTHEQUE".Mobile[#index].Pos[0].Entr0_Ap_Pos[0] := "I_RPO_TRS57";
	"DB_BIBLIOTHEQUE".Mobile[#index].Pos[0].Entr1_Ap_Pos[0] := "I_RPF_TRS57";
	"DB_BIBLIOTHEQUE".Mobile[#index].Pos[0].Sort0[0] := "I_CO_TRS57";
	"DB_BIBLIOTHEQUE".Mobile[#index].Pos[0].Sort0_Pr_Fin_Pos[0] := "I_CO_TRS57";

	//position ouverture
	"DB_BIBLIOTHEQUE".Mobile[#index].Pos[1].Entr0_Ap_Pos[0] := "I_RPF_TRS57";
	"DB_BIBLIOTHEQUE".Mobile[#index].Pos[1].Entr1_Ap_Pos[0] := "I_RPO_TRS57";
	"DB_BIBLIOTHEQUE".Mobile[#index].Pos[1].Sort1[0] := "I_CO_TRS57";
	"DB_BIBLIOTHEQUE".Mobile[#index].Pos[1].Sort0_Pr_Fin_Pos[0] := "I_CO_TRS57";
	#index := #index + 1;
	//++++++++++++++++++++++++++++++++++++++++++++++++++++++++++++++/*365*/
	"DB_BIBLIOTHEQUE".Mobile[#index].Nom := 'EXT2_S58';
	"DB_BIBLIOTHEQUE".Mobile[#index].Tjr_Desasservi := TRUE;
	"DB_BIBLIOTHEQUE".Mobile[#index].Pos[0].Nom := 'DROIT';
	"Init_Tps"(#index);

	//position fermeture
	"DB_BIBLIOTHEQUE".Mobile[#index].Pos[0].Entr0_Ap_Pos[0] := "I_RPO_TRS58";
	"DB_BIBLIOTHEQUE".Mobile[#index].Pos[0].Entr1_Ap_Pos[0] := "I_RPF_TRS58";
	"DB_BIBLIOTHEQUE".Mobile[#index].Pos[0].Sort0[0] := "I_CO_TRS58";
	"DB_BIBLIOTHEQUE".Mobile[#index].Pos[0].Sort0_Pr_Fin_Pos[0] := "I_CO_TRS58";

	//position ouverture
	"DB_BIBLIOTHEQUE".Mobile[#index].Pos[1].Entr0_Ap_Pos[0] := "I_RPF_TRS58";
	"DB_BIBLIOTHEQUE".Mobile[#index].Pos[1].Entr1_Ap_Pos[0] := "I_RPO_TRS58";
	"DB_BIBLIOTHEQUE".Mobile[#index].Pos[1].Sort1[0] := "I_CO_TRS58";
	"DB_BIBLIOTHEQUE".Mobile[#index].Pos[1].Sort0_Pr_Fin_Pos[0] := "I_CO_TRS58";
	#index := #index + 1;
	//++++++++++++++++++++++++++++++++++++++++++++++++++++++++++++++/*366*/
	"DB_BIBLIOTHEQUE".Mobile[#index].Nom := 'EXT2_S30';
	"DB_BIBLIOTHEQUE".Mobile[#index].Tjr_Desasservi := TRUE;
	"DB_BIBLIOTHEQUE".Mobile[#index].Pos[0].Nom := 'DROIT';
	"Init_Tps"(#index);

	//position fermeture
	"DB_BIBLIOTHEQUE".Mobile[#index].Pos[0].Entr0_Ap_Pos[0] := "I_RPO_EXT2_S30";
	"DB_BIBLIOTHEQUE".Mobile[#index].Pos[0].Entr1_Ap_Pos[0] := "I_RPF_EXT2_S30";
	"DB_BIBLIOTHEQUE".Mobile[#index].Pos[0].Sort0[0] := "I_CO_TRS30";
	"DB_BIBLIOTHEQUE".Mobile[#index].Pos[0].Sort0_Pr_Fin_Pos[0] := "I_CO_TRS30";

	//position ouverture
	"DB_BIBLIOTHEQUE".Mobile[#index].Pos[1].Entr0_Ap_Pos[0] := "I_RPF_EXT2_S30";
	"DB_BIBLIOTHEQUE".Mobile[#index].Pos[1].Entr1_Ap_Pos[0] := "I_RPO_EXT2_S30";
	"DB_BIBLIOTHEQUE".Mobile[#index].Pos[1].Sort1[0] := "I_CO_TRS30";
	"DB_BIBLIOTHEQUE".Mobile[#index].Pos[1].Sort0_Pr_Fin_Pos[0] := "I_CO_TRS30";
	#index := #index + 1;
	//++++++++++++++++++++++++++++++++++++++++++++++++++++++++++++++/*367*/
	"DB_BIBLIOTHEQUE".Mobile[#index].Nom := 'EXT2_S33';
	"DB_BIBLIOTHEQUE".Mobile[#index].Tjr_Desasservi := TRUE;
	"DB_BIBLIOTHEQUE".Mobile[#index].Pos[0].Nom := 'DROIT';
	"Init_Tps"(#index);

	//position fermeture
	"DB_BIBLIOTHEQUE".Mobile[#index].Pos[0].Entr0_Ap_Pos[0] := "I_RPO_EXT2_S33";
	"DB_BIBLIOTHEQUE".Mobile[#index].Pos[0].Entr1_Ap_Pos[0] := "I_RPF_EXT2_S33";
	"DB_BIBLIOTHEQUE".Mobile[#index].Pos[0].Sort0[0] := "I_CO_TRS33";
	"DB_BIBLIOTHEQUE".Mobile[#index].Pos[0].Sort0_Pr_Fin_Pos[0] := "I_CO_TRS33";

	//position ouverture
	"DB_BIBLIOTHEQUE".Mobile[#index].Pos[1].Entr0_Ap_Pos[0] := "I_RPF_EXT2_S33";
	"DB_BIBLIOTHEQUE".Mobile[#index].Pos[1].Entr1_Ap_Pos[0] := "I_RPO_EXT2_S33";
	"DB_BIBLIOTHEQUE".Mobile[#index].Pos[1].Sort1[0] := "I_CO_TRS33";
	"DB_BIBLIOTHEQUE".Mobile[#index].Pos[1].Sort0_Pr_Fin_Pos[0] := "I_CO_TRS33";
	#index := #index + 1;
	//++++++++++++++++++++++++++++++++++++++++++++++++++++++++++++++/*368*/
	"DB_BIBLIOTHEQUE".Mobile[#index].Nom := 'EXT2_S36';
	"DB_BIBLIOTHEQUE".Mobile[#index].Tjr_Desasservi := TRUE;
	"DB_BIBLIOTHEQUE".Mobile[#index].Pos[0].Nom := 'DROIT';
	"Init_Tps"(#index);

	//position fermeture
	"DB_BIBLIOTHEQUE".Mobile[#index].Pos[0].Entr0_Ap_Pos[0] := "I_RPO_EXT2_S36";
	"DB_BIBLIOTHEQUE".Mobile[#index].Pos[0].Entr1_Ap_Pos[0] := "I_RPF_EXT2_S36";
	"DB_BIBLIOTHEQUE".Mobile[#index].Pos[0].Sort0[0] := "I_CO_TRS36";
	"DB_BIBLIOTHEQUE".Mobile[#index].Pos[0].Sort0_Pr_Fin_Pos[0] := "I_CO_TRS36";

	//position ouverture
	"DB_BIBLIOTHEQUE".Mobile[#index].Pos[1].Entr0_Ap_Pos[0] := "I_RPF_EXT2_S36";
	"DB_BIBLIOTHEQUE".Mobile[#index].Pos[1].Entr1_Ap_Pos[0] := "I_RPO_EXT2_S36";
	"DB_BIBLIOTHEQUE".Mobile[#index].Pos[1].Sort1[0] := "I_CO_TRS36";
	"DB_BIBLIOTHEQUE".Mobile[#index].Pos[1].Sort0_Pr_Fin_Pos[0] := "I_CO_TRS36";
	#index := #index + 1;
	//++++++++++++++++++++++++++++++++++++++++++++++++++++++++++++++/*369*/
	"DB_BIBLIOTHEQUE".Mobile[#index].Nom := 'VFR1';
	"DB_BIBLIOTHEQUE".Mobile[#index].Pos[0].Nom := 'MARCHE';
	"DB_BIBLIOTHEQUE".Mobile[#index].Tjr_Desasservi := TRUE;
	"Init_Tps"(#index);

	// Entrées avant pos
	"DB_BIBLIOTHEQUE".Mobile[#index].Pos[0].Entr0_Av_Pos[0] := "I_RD_DISJ_VFR1";

	// Entrées apres pos
	"DB_BIBLIOTHEQUE".Mobile[#index].Pos[0].Entr0_Ap_Pos[1] := "I_RD_DISJ_VFR1";
	"DB_BIBLIOTHEQUE".Mobile[#index].Pos[0].Entr1_Ap_Pos[0] := "I_RM_VFR1";

	// Entrées fin pos
	"DB_BIBLIOTHEQUE".Mobile[#index].Pos[0].Entr0_Ap_Fin_Pos[0] := "I_RM_VFR1";

	// Sorties
	"DB_BIBLIOTHEQUE".Mobile[#index].Pos[0].Sort1[0] := "I_CM_VFR1";
	"DB_BIBLIOTHEQUE".Mobile[#index].Pos[0].Sort0_Pr_Fin_Pos[0] := "I_CM_VFR1";
	#index := #index + 1;
	//++++++++++++++++++++++++++++++++++++++++++++++++++++++++++++++/*370*/
	"DB_BIBLIOTHEQUE".Mobile[#index].Nom := 'FR1';
	"DB_BIBLIOTHEQUE".Mobile[#index].Pos[0].Nom := 'MARCHE';
	"DB_BIBLIOTHEQUE".Mobile[#index].Tjr_Desasservi := TRUE;
	"Init_Tps"(#index);

	// Entrées fin pos
	"DB_BIBLIOTHEQUE".Mobile[#index].Pos[0].Entr0_Ap_Fin_Pos[0] := "I_RM_FR1";

	// Sorties
	"DB_BIBLIOTHEQUE".Mobile[#index].Pos[0].Sort1[0] := "I_CM_FR1";
	"DB_BIBLIOTHEQUE".Mobile[#index].Pos[0].Sort0_Pr_Fin_Pos[0] := "I_CM_FR1";
	#index := #index + 1;
	//++++++++++++++++++++++++++++++++++++++++++++++++++++++++++++++/*371*/
	"DB_BIBLIOTHEQUE".Mobile[#index].Nom := 'VAFR1';
	"DB_BIBLIOTHEQUE".Mobile[#index].Pos[0].Nom := 'FERMETURE';
	"DB_BIBLIOTHEQUE".Mobile[#index].Pos[1].Nom := 'OUVERTURE';
	"DB_BIBLIOTHEQUE".Mobile[#index].Tjr_Desasservi := TRUE;
	"Init_Tps"(#index);

	//position fermeture
	"DB_BIBLIOTHEQUE".Mobile[#index].Pos[0].Entr0_Ap_Pos[0] := "I_RPO_VAFR1";
	"DB_BIBLIOTHEQUE".Mobile[#index].Pos[0].Entr1_Ap_Pos[0] := "I_RPF_VAFR1";
	"DB_BIBLIOTHEQUE".Mobile[#index].Pos[0].Sort0[0] := "I_CMAV_VAFR1";
	"DB_BIBLIOTHEQUE".Mobile[#index].Pos[0].Sort0_Pr_Fin_Pos[0] := "I_CMAV_VAFR1";

	//position ouverture
	"DB_BIBLIOTHEQUE".Mobile[#index].Pos[1].Entr0_Ap_Pos[0] := "I_RPF_VAFR1";
	"DB_BIBLIOTHEQUE".Mobile[#index].Pos[1].Entr1_Ap_Pos[0] := "I_RPO_VAFR1";
	"DB_BIBLIOTHEQUE".Mobile[#index].Pos[1].Sort1[0] := "I_CMAV_VAFR1";
	"DB_BIBLIOTHEQUE".Mobile[#index].Pos[1].Sort0_Pr_Fin_Pos[0] := "I_CMAV_VAFR1";
	#index := #index + 1;
	//++++++++++++++++++++++++++++++++++++++++++++++++++++++++++++++/**/

END_FUNCTION

